TYPE
    TcoCustomTimeStruct :
    STRUCT
        Year : WORD;
        Month : WORD;

        Day : WORD;
        Hour : WORD;
        Minute : WORD;
        Second : WORD;
        Milliseconds : WORD;
    END_STRUCT
END_TYPE

(* stored: Version 1.1.0.1
   DUT TcoCustomTimeStruct: Id {c752a31a-4b9c-4ade-a760-f62e46f31888} *)
